KUKA KRL program: chk_w4_grp1_clo.src

&ACCESS RVO2
&COMMENT Check GRP Z1 ACCELO CLOSE
DEF chk_w4_grp1_clo( )

; Check gripper accelo CLOSE Z1.1/2/3/4/5
;//---- Start User-------

$TIMER[10] = 0
$TIMER_STOP[10] = FALSE

WAIT FOR ($IN[38] AND $IN[40] AND $IN[42] AND $IN[44] AND $IN[46])
WAIT FOR (NOT $IN[37] AND NOT $IN[39] AND NOT $IN[43] AND NOT $IN[45])

$TIMER_STOP[10] = TRUE
$TIMER[10] = 0

;//---- End User---------

END
